{attribute 'hide_all_locals'}
FUNCTION_BLOCK PUBLIC ABSTRACT FB_Employee_1 IMPLEMENTS I_Employee_1
VAR_INPUT
END_VAR
VAR_OUTPUT
END_VAR
VAR
	nPersonnelNumberBacking :	UINT;
	sFirstNameBacking		:	STRING;
	sLastNameBacking		:	STRING;
END_VAR

METHOD PUBLIC GetFullName : STRING
VAR_INPUT
END_VAR
GetFullName := CONCAT(CONCAT(CONCAT(CONCAT(TO_STRING(nPersonnelNumber), ': '), sFirstName), ' '), sLastName);
END_METHOD

METHOD PUBLIC ABSTRACT GetMonthlySalary : LREAL
VAR_INPUT
END_VAR
END_METHOD

{attribute 'monitoring' := 'variable'}
PROPERTY PUBLIC nPersonnelNumber : UINT
GET
nPersonnelNumber := nPersonnelNumberBacking;
END_GET
SET
nPersonnelNumberBacking := nPersonnelNumber;
END_SET
END_PROPERTY

{attribute 'monitoring' := 'variable'}
PROPERTY PUBLIC sFirstName : STRING
GET
sFirstName := sFirstNameBacking;
END_GET
SET
sFirstNameBacking := sFirstName;
END_SET
END_PROPERTY

{attribute 'monitoring' := 'variable'}
PROPERTY PUBLIC sLastName : STRING
GET
sLastName := sLastNameBacking;
END_GET
SET
sLastNameBacking := sLastName;
END_SET
END_PROPERTY

END_FUNCTION_BLOCK

(* stored: Version 1.1.0.1, ProductVersion 3.1.4024.12
   POU FB_Employee_1: Id {6457be40-59c8-4808-b942-97fc7dfcdf69}, SpecialFunc None
   Method GetFullName: Id {23dec1ff-9ffa-41bd-b34c-aa2b8148499b}
   Method GetMonthlySalary: Id {d9a3ae75-55a5-4ba4-8096-352ec7d0118d}
   Property nPersonnelNumber: Id {ca35b716-9316-4ac5-a483-363d3f6f8d95}
   Get Get: Id {1f8d65b6-a3a5-4864-9561-584b659cde32}
   Set Set: Id {c77b21f5-0e83-47d0-b8c9-df3b029cf132}
   Property sFirstName: Id {cb96c46e-6697-4ee8-9be9-4405fb953d06}
   Get Get: Id {8cf9f14d-a12b-4d65-88aa-1965682651c1}
   Set Set: Id {c5459749-aad0-45e3-9435-cf39ee597117}
   Property sLastName: Id {b5e1b7f0-a6db-4df4-a404-ecdbe2412e11}
   Get Get: Id {0e328a25-766a-4e02-9bde-edeb61c794dc}
   Set Set: Id {367abf85-df4b-4da9-9b37-3e0dbf5ac2c6} *)
